{attribute 'linkalways'} 
{attribute 'no_explicit_call' := 'This FB is a CLASS and must be accessed using methods or properties'}
{attribute 'enable_dynamic_creation'}
FUNCTION_BLOCK GetPaginatedBlueprintsVisitor IMPLEMENTS I_NodeFactoryVisitor, I_NodePrototypeVisitor, I_NodeVisitor, I_ExtensionVisitor, I_InputPortVisitor, I_OutputPortVisitor, I_MetadataVisitor, I_ContentVisitor, I_ParameterVisitor, I_AlarmVisitor
VAR
	serializer : I_Serializer;
	offset : UDINT;
	maxLimit : UDINT;
	
	// used to track count
	currentIndex : UDINT;
	endIndex : UDINT;
	blueprintsCollected : UDINT;
	totalBlueprints : UDINT;
END_VAR

METHOD PUBLIC Initialize
VAR_INPUT
	Serializer : I_Serializer;
	Offset : UDINT;
	MaxLimit : UDINT;
END_VAR
THIS^.serializer := Serializer;
THIS^.offset := Offset;
THIS^.maxLimit := MaxLimit;

THIS^.currentIndex := 0;
THIS^.endIndex := Offset + MaxLimit -1;

THIS^.blueprintsCollected := 0;
THIS^.totalBlueprints := 0;
END_METHOD

METHOD VisitAlarm
VAR_INPUT
	VisitingAlarm : I_Alarm;
END_VAR
serializer.AddString(VisitingAlarm.Message);
END_METHOD

METHOD VisitContent
VAR_INPUT
	VisitingContent : I_Content;
END_VAR
serializer.StartObject();

serializer.AddKeyString('name', VisitingContent.Name);
serializer.Addkey('datatype');
VisitingContent.Data.SerializeTypeWith(serializer);

IF VisitingContent.Metadatum.HasMetadata THEN
	serializer.addkey('metadata');
	serializer.StartArray();
	VisitingContent.Metadatum.Accept(THIS^);
	serializer.EndArray();
END_IF

serializer.EndObject();
END_METHOD

METHOD VisitExtension
VAR_INPUT
	VisitingExtension : I_Extension;
END_VAR
Serializer.StartObject();
Serializer.AddKeyString('name', VisitingExtension.Name);

IF VisitingExtension.Metadatum.HasMetadata THEN
	serializer.addkey('metadata');
	serializer.StartArray();
	VisitingExtension.Metadatum.Accept(THIS^);
	serializer.EndArray();
END_IF

IF VisitingExtension.Alarms.HasAlarms THEN
	serializer.addkey('alarms');
	serializer.StartArray();
	VisitingExtension.Alarms.Accept(THIS^);
	serializer.EndArray();
END_IF

IF VisitingExtension.InputPorts.HasInputPorts THEN
	serializer.addkey('inputPorts');
	serializer.StartArray();
	VisitingExtension.InputPorts.Accept(THIS^);
	serializer.EndArray();
END_IF

IF VisitingExtension.OutputPorts.HasOutputPorts THEN
	serializer.addkey('outputPorts');
	serializer.StartArray();
	VisitingExtension.OutputPorts.Accept(THIS^);
	serializer.EndArray();
END_IF

IF VisitingExtension.Parameters.HasParameters THEN
	serializer.addkey('parameters');
	serializer.StartArray();
	VisitingExtension.Parameters.Accept(THIS^);
	serializer.EndArray();
END_IF

IF VisitingExtension.Contents.HasContents THEN
	serializer.addkey('contents');
	serializer.StartArray();
	VisitingExtension.Contents.Accept(THIS^);
	serializer.EndArray();
END_IF

Serializer.EndObject();
END_METHOD

METHOD VisitInputPort
VAR_INPUT
	VisitingInputPort : I_InputPort;
END_VAR
serializer.StartObject();

serializer.AddKeyString('name', VisitingInputPort.Name);
serializer.Addkey('datatype');
VisitingInputPort.Data.SerializeTypeWith(serializer);

IF VisitingInputPort.Metadatum.HasMetadata THEN
	serializer.addkey('metadata');
	serializer.StartArray();
	VisitingInputPort.Metadatum.Accept(THIS^);
	serializer.EndArray();
END_IF

serializer.EndObject();
END_METHOD

METHOD VisitMetadatum
VAR_INPUT
	VisitingMetadatum : I_Metadata;
END_VAR
serializer.StartObject();
serializer.AddKeyString('name', VisitingMetadatum.Name);
serializer.AddkeyObject('value', VisitingMetadatum.Data);
serializer.EndObject();
END_METHOD

METHOD VisitNode
VAR_INPUT
	VisitingNode : I_Node;
END_VAR
serializer.StartObject();

IF VisitingNode.Metadatum.HasMetadata THEN
	serializer.addkey('metadata');
	serializer.StartArray();
	VisitingNode.Metadatum.Accept(THIS^);
	serializer.EndArray();
END_IF

IF VisitingNode.Alarms.HasAlarms THEN
	serializer.addkey('alarms');
	serializer.StartArray();
	VisitingNode.Alarms.Accept(THIS^);
	serializer.EndArray();
END_IF

IF VisitingNode.Extensions.HasExtensions THEN
	serializer.addkey('extensions');
	serializer.StartArray();
	VisitingNode.Extensions.Accept(THIS^);
	serializer.EndArray();
END_IF

IF VisitingNode.InputPorts.HasInputPorts THEN
	serializer.addkey('inputPorts');
	serializer.StartArray();
	VisitingNode.InputPorts.Accept(THIS^);
	serializer.EndArray();
END_IF

IF VisitingNode.OutputPorts.HasOutputPorts THEN
	serializer.addkey('outputPorts');
	serializer.StartArray();
	VisitingNode.OutputPorts.Accept(THIS^);
	serializer.EndArray();
END_IF

IF VisitingNode.Parameters.HasParameters THEN
	serializer.addkey('parameters');
	serializer.StartArray();
	VisitingNode.Parameters.Accept(THIS^);
	serializer.EndArray();
END_IF

IF VisitingNode.Contents.HasContents THEN
	serializer.addkey('contents');
	serializer.StartArray();
	VisitingNode.Contents.Accept(THIS^);
	serializer.EndArray();
END_IF

serializer.EndObject();
END_METHOD

METHOD VisitNodeFactory
VAR_INPUT
	VisitingNodeFactory : I_NodeFactory;
END_VAR
serializer.StartObject();
serializer.AddKey('blueprints');
serializer.StartArray();
VisitingNodeFactory.NodePrototypes.Accept(THIS^);
serializer.EndArray();
serializer.AddKeyUdint('returnedCount', blueprintsCollected);
serializer.AddKeyUdint('totalCount', totalBlueprints);
serializer.AddKeyUdint('nextOffset', offset + blueprintsCollected);
serializer.AddKeyBool('hasMore', offset + blueprintsCollected < totalBlueprints); 
serializer.EndObject();
END_METHOD

METHOD VisitNodePrototype
VAR_INPUT
	VisitingPrototype : I_NodePrototype;
END_VAR
// we're not yet in range of collection
IF currentIndex < offset THEN
	currentIndex := currentIndex + 1;
	totalBlueprints := totalBlueprints + 1;
	RETURN;
END_IF

// we're over range of the collection
IF currentIndex > endIndex THEN
	currentIndex := currentIndex + 1;
	totalBlueprints := totalBlueprints + 1;
	RETURN;
END_IF

// we're in the range to collect. 

blueprintsCollected := blueprintsCollected + 1;
currentIndex := currentIndex + 1;
totalBlueprints := totalBlueprints + 1;

serializer.StartObject();
serializer.AddKeyString('path', VisitingPrototype.Path);
serializer.AddKey('node');
VisitingPrototype.Node.Accept(THIS^);
serializer.EndObject();
END_METHOD

METHOD VisitOutputPort
VAR_INPUT
	VisitingOutputPort : I_OutputPort;
END_VAR
serializer.StartObject();

serializer.AddKeyString('name', VisitingOutputPort.Name);
serializer.Addkey('datatype');
VisitingOutputPort.Data.SerializeTypeWith(serializer);

IF VisitingOutputPort.Metadatum.HasMetadata THEN
	serializer.addkey('metadata');
	serializer.StartArray();
	VisitingOutputPort.Metadatum.Accept(THIS^);
	serializer.EndArray();
END_IF

serializer.EndObject();
END_METHOD

METHOD VisitParameter
VAR_INPUT
	VisitingProperty : I_Parameter;
END_VAR
serializer.StartObject();

serializer.AddKeyString('name', VisitingProperty.Name);
serializer.Addkey('datatype');
VisitingProperty.Data.SerializeTypeWith(serializer);
serializer.Addkey('defaultValue');
VisitingProperty.Data.SerializeWith(serializer);

IF VisitingProperty.Metadatum.HasMetadata THEN
	serializer.addkey('metadata');
	serializer.StartArray();
	VisitingProperty.Metadatum.Accept(THIS^);
	serializer.EndArray();
END_IF

Serializer.EndObject();
END_METHOD

END_FUNCTION_BLOCK

(* stored: Version 1.1.0.1, ProductVersion 3.1.4024.13
   POU GetPaginatedBlueprintsVisitor: Id {7e8b6503-4c5b-0b40-34cf-a29cc72bbf42}, SpecialFunc None
   Method Initialize: Id {4ffc1cf6-703e-0a49-2998-b227262fb33a}
   Method VisitAlarm: Id {f2f44703-628c-0228-1867-5201faebe8a4}
   Method VisitContent: Id {949aebd3-b860-0900-15b0-53c0f5d9719d}
   Method VisitExtension: Id {2cd717cb-a98c-06a4-0d23-072d8ffe6668}
   Method VisitInputPort: Id {783644e7-394d-0b08-398e-b64e4740f305}
   Method VisitMetadatum: Id {b9eb07fa-4802-0ba8-3506-3e36d2e825a0}
   Method VisitNode: Id {de998030-02f5-0231-15fa-0722a28b6764}
   Method VisitNodeFactory: Id {a3611590-b2a2-0475-18bc-70a4df530f86}
   Method VisitNodePrototype: Id {52a611cd-0fa0-0658-13cb-2406718fa138}
   Method VisitOutputPort: Id {8c21d527-3d65-0998-3377-cd368c70270e}
   Method VisitParameter: Id {202e004f-4a7d-0025-2c3f-ea7bf62d6015} *)
